PROGRAM P_Demo_FB_DALIV2OnAndStepUp
VAR
    fbFB_DALIV2OnAndStepUp        : FB_DALIV2OnAndStepUp;
    stCommandBuffer : ST_DALIV2CommandBuffer;

    bTrigger        : BOOL;
    nLampAddr        : BYTE := 0;


    bBusy           : BOOL;
    bErr            : BOOL;
    nErrId          : UDINT;
END_VAR

// =============================================================================
// 场景：面板加亮按钮的开灯兼调光实现：灯关时按一下就开（且渐亮）；灯亮时按一下递增。...
//
// 价值：DALI 协议标准命令的轻量封装。
//
// 验证步骤：
//   1. 通信 FB 跑起；编译；登录。
//   2. 在线 bTrigger 一次上升沿；等 bBusy 回 FALSE。
//   3. 观察 short addr 0 灯的物理亮度变化是否符合本命令描述。
// =============================================================================
fbFB_DALIV2OnAndStepUp(
    bStart           := bTrigger,
    nAddr            := nLampAddr,
    eAddrType        := eDALIV2AddrTypeShort,
    eCommandPriority := eDALIV2CommandPriorityMiddle,
    stCommandBuffer  := stCommandBuffer
);

bBusy  := fbFB_DALIV2OnAndStepUp.bBusy;
bErr   := fbFB_DALIV2OnAndStepUp.bError;
nErrId := fbFB_DALIV2OnAndStepUp.nErrorId;

END_PROGRAM

(* stored: Version 1.1.0.1, ProductVersion 3.1.4024.5
   POU P_Demo_FB_DALIV2OnAndStepUp: Id {2c83b6d6-dda8-5e2d-8926-beae861ecb70}, SpecialFunc None *)
